// TIA Portal V17 export
// export: Created 2023-03-08T16:44:23.1874801Z, ExportSetting None, DisplayName Totally Integrated Automation Portal, DisplayVersion V17 Update 4, DisplayName TIA Portal Openness, DisplayVersion V17 Update 4, DisplayName TIA Portal Version Control Interface, DisplayVersion V17, DisplayName STEP 7 Professional, DisplayVersion V17 Update 4, DisplayName STEP 7 Safety, DisplayVersion V17, DisplayName WinCC Advanced / Unified PC, DisplayVersion V17 Update 4
DATA_BLOCK "DI"   // DB12
{ S7_Optimized_Access := 'TRUE' }
// stored: AutoNumber false, MemoryReserve 100
   VAR
      LS_045200 : Bool;   // SEPARATOR SUCTION SIDE 1ST. STAGE VERY HIGH LEVEL
      LS_045201 : Bool;   // SEPARATOR SUCTION SIDE 1ST. STAGE VERY LOW LEVEL
      LS_045210 : Bool;   // SEPARATOR DISCHARGE SIDE 1ST. STAGE VERY HIGH
      LS_045211 : Bool;   // SEPARATOR DISCHARGE SIDE 1ST. STAGE VERY LOW
      LS_045220 : Bool;   // SEPARATOR DISCHARGE SIDE 2ND STAGE VERY HIGH
      LS_045221 : Bool;   // SEPARATOR DISCHARGE SIDE 2ND STAGE VERY LOW
      LS_045230 : Bool;   // COALESCER DISCHARGE SIDE 3RD STAGE VERY HIGH
      LS_045232 : Bool;   // COALESCER DISCHARGE SIDE 3RD STAGE VERY LOW
      LS_045240 : Bool;   // OUTLET COALESCER DISCHARGE SIDE 3RD STAGE VERY HIGH
      LS_045242 : Bool;   // OUTLET COALESCER DISCHARGE SIDE 3RD STAGE VERY LOW
      GS_045405 : Bool;   // FLYWHEEL COVER CLOSED
      HS_045009 : Bool;   // EMERGENCY STOP FROM LCP
      HS_045501 : Bool;   // EMERGENCY STOP FROM UCP
      XY_045037 : Bool;   // PROCESS SHUTDOWN FROM DCS
      XY_045035 : Bool;   // EXTERNAL TRIP FROM ESD
      XY_045036 : Bool;   // GAS DETECTION FROM ESD
      LS_045574 : Bool;   // HYDRAULIC OIL VESSEL LOW LEVEL
      LS_045305 : Bool;   // LUBE OIL IN CRANKCASE LOW LEVEL
      LS_045426 : Bool;   // DOWNSTREAM FLOW HEATER LOW LEVEL
      GSH_045206 : Bool;   // BYPASS CONTROL VALVE OVER 1ST-3RD STAGE OPEN
      GSH_045203 : Bool;   // CONDENSATE DRAIN VALVE SEPARATOR SUCTION SIDE 1ST STAGE OPEN
      GSL_045203 : Bool;   // CONDENSATE DRAIN VALVE SEPARATOR SUCTION SIDE 1ST STAGE CLOSED
      GSH_045204 : Bool;   // CONDENSATE DRAIN VALVE SEPARATOR DISCHARGE SIDE 1ST STAGE OPEN
      GSL_045204 : Bool;   // CONDENSATE DRAIN VALVE SEPARATOR DISCHARGE SIDE 1ST STAGE CLOSED
      GSH_045205 : Bool;   // CONDENSATE DRAIN VALVE SEPARATOR DISCHARGE SIDE 2ND STAGE OPEN
      GSL_045205 : Bool;   // CONDENSATE DRAIN VALVE SEPARATOR DISCHARGE SIDE 2ND STAGE CLOSED
      GSH_045207A : Bool;   // CONDENSATE DRAIN VALVE SEPARATOR DISCHARGE SIDE 2ND STAGE OPEN
      GSL_045207A : Bool;   // CONDENSATE DRAIN VALVE SEPARATOR DISCHARGE SIDE 2ND STAGE CLOSED
      GSH_045207B : Bool;   // CONDENSATE DRAIN VALVE SEPARATOR DISCHARGE SIDE 2ND STAGE OPEN
      GSL_045207B : Bool;   // CONDENSATE DRAIN VALVE SEPARATOR DISCHARGE SIDE 2ND STAGE CLOSED
      GSH_045208A : Bool;   // CONDENSATE DRAIN VALVE SEPARATOR DISCHARGE SIDE 3RD STAGE OPEN
      GSL_045208A : Bool;   // CONDENSATE DRAIN VALVE SEPARATOR DISCHARGE SIDE 3RD STAGE CLOSED
      GSH_045208B : Bool;   // CONDENSATE DRAIN VALVE SEPARATOR DISCHARGE SIDE 3RD STAGE OPEN
      GSL_045208B : Bool;   // CONDENSATE DRAIN VALVE SEPARATOR DISCHARGE SIDE 3RD STAGE CLOSED
      TS_045307 : Bool;   // LUBE OIL IN CRANKCASE TEMPERATURE LIMITER
      TC_045306 : Bool;   // LUBE OIL IN CRANKCASE TEMPERATURE CONTROLLER
      TS_045428 : Bool;   // COOLING WATER HEATER TEMPERATURE LIMITER
      TC_045427 : Bool;   // COOLING WATER HEATER TEMPERATURE CONTROLLER
      HS_045001 : Bool;   // COMPRESSOR PREPARE TO START FROM LCP
      HS_045002A : Bool;   // COMPRESSOR PROCESS GAS MODE START FROM LCP
      HS_045002B : Bool;   // COMPRESSOR PROCESS GAS MODE STOP FROM LCP
      HS_045003A : Bool;   // COMPRESSOR NITROGEN MODE START FROM LCP
      HS_045003B : Bool;   // COMPRESSOR NITROGEN MODE STOP FROM LCP
      HS_045004A : Bool;   // CRANKCASE LUBE OIL HEATER START FROM LCP
      HS_045004B : Bool;   // CRANKCASE LUBE OIL HEATER STOP FROM LCP
      HS_045005A : Bool;   // ELECTRICAL OIL PUMP START FROM LCP
      HS_045005B : Bool;   // ELECTRICAL OIL PUMP STOP FROM LCP
      HS_045006A : Bool;   // HYDROCOM HYDRAULIC PUMP START FROM LCP
      HS_045006B : Bool;   // HYDROCOM HYDRAULIC PUMP STOP FROM LCP
      HS_045007A : Bool;   // COMPRESSOR REMOTE FROM LCP
      HS_045007B : Bool;   // COMPRESSOR LOCAL FROM LCP
      HS_045008 : Bool;   // FAULT RESET FROM LCP
      HS_045010 : Bool;   // LAMP TEST FROM LCP
      HS_045011A : Bool;   // COOLANT HEATER START FROM LCP
      HS_045011B : Bool;   // COOLANT HEATER STOP FROM LCP
      HS_045012A : Bool;   // COOLANT PUMP 1 START FROM LCP
      HS_045012B : Bool;   // COOLANT PUMP 1 STOP FROM LCP
      HS_045013A : Bool;   // COOLANT PUMP 2 START FROM LCP
      HS_045013B : Bool;   // COOLANT PUMP 2 STOP FROM LCP
      HS_045014A : Bool;   // FAN 1 START FROM LCP
      HS_045014B : Bool;   // FAN 1 STOP FROM LCP
      HS_045015A : Bool;   // FAN 2 START FROM LCP
      HS_045015B : Bool;   // FAN 2 STOP FROM LCP
      HS_045018A : Bool;   // LOUVER 1 OPEN FROM LCP
      HS_045018B : Bool;   // LOUVER 1 CLOSE FROM LCP
      HS_045019A : Bool;   // LOUVER 2 OPEN FROM LCP
      HS_045019B : Bool;   // LOUVER 2 CLOSE FROM LCP
      HS_045020A : Bool;   // LOUVER 3 OPEN FROM LCP
      HS_045020B : Bool;   // LOUVER 3 CLOSE FROM LCP
      HS_045021A : Bool;   // LOUVER 4 OPEN FROM LCP
      HS_045021B : Bool;   // LOUVER 4 CLOSE FROM LCP
      GSH_045544 : Bool;   // LOUVER 1 OPEN
      GSL_045544 : Bool;   // LOUVER 1 CLOSED
      GSH_045545 : Bool;   // LOUVER 2 OPEN
      GSL_045545 : Bool;   // LOUVER 2 CLOSED
      GSH_045546 : Bool;   // LOUVER 3 OPEN
      GSL_045546 : Bool;   // LOUVER 3 CLOSED
      GSH_045547 : Bool;   // LOUVER 4 OPEN
      GSL_045547 : Bool;   // LOUVER 4 CLOSED
      XY_045001 : Bool;   // OIL HEATER RUNNING FEEDBACK FROM MCC
      XY_045002 : Bool;   // OIL HEATER FAULT FEEDBACK FROM MCC
      XY_045003 : Bool;   // AUXILIARY OIL PUMP RUNNING FEEDBACK FROM MCC
      XY_045004 : Bool;   // AUXILIARY OIL PUMP FAULT FEEDBACK FROM MCC
      XY_045005 : Bool;   // HYDROCOM HYDRAULIC PUMP RUNNING FEEDBACK FROM MCC
      XY_045006 : Bool;   // HYDROCOM HYDRAULIC PUMP FAULT FEEDBACK FROM MCC
      XY_045007 : Bool;   // COOLANT HEATER RUNNING FEEDBACK FROM MCC
      XY_045008 : Bool;   // COOLANT HEATER FAULT FEEDBACK FROM MCC
      XY_045009 : Bool;   // COOLANT PUMP 1 RUNNING FEEDBACK FROM MCC
      XY_045010 : Bool;   // COOLANT PUMP 1 FAULT FEEDBACK FROM MCC
      XY_045011 : Bool;   // COOLANT PUMP 2 RUNNING FEEDBACK FROM MCC
      XY_045012 : Bool;   // COOLANT PUMP 2 FAULT FEEDBACK FROM MCC
      XY_045013 : Bool;   // FAN 1 MOTOR RUNNING FEEDBACK FROM MCC
      XY_045014 : Bool;   // FAN 1 MOTOR FAULT FEEDBACK FROM MCC
      XY_045015 : Bool;   // FAN 2 MOTOR RUNNING FEEDBACK FROM MCC
      XY_045016 : Bool;   // FAN 2 MOTOR FAULT FEEDBACK FROM MCC
      XY_045021 : Bool;   // LOUVER 1 MOTOR RUNNING FEEDBACK FROM MCC
      XY_045022 : Bool;   // LOUVER 1 MOTOR FAULT FEEDBACK FROM MCC
      XY_045023 : Bool;   // LOUVER 2 MOTOR RUNNING FEEDBACK FROM MCC
      XY_045024 : Bool;   // LOUVER 2 MOTOR FAULT FEEDBACK FROM MCC
      XY_045025 : Bool;   // LOUVER 3 MOTOR RUNNING FEEDBACK FROM MCC
      XY_045026 : Bool;   // LOUVER 3 MOTOR FAULT FEEDBACK FROM MCC
      XY_045027 : Bool;   // LOUVER 4 MOTOR RUNNING FEEDBACK FROM MCC
      XY_045028 : Bool;   // LOUVER 4 MOTOR FAULT FEEDBACK FROM MCC
      XY_045029 : Bool;   // COMPRESSOR RUNNING FEEDBACK FROM MV-MCC
      XY_045030 : Bool;   // COMPRESSOR FAULT FEEDBACK FROM MV-MCC
      FS_045540 : Bool;   // AIR OUTLET NOISE ENCLOSURE LOW FLOW
      FS_045541 : Bool;   // AIR OUTLET NOISE ENCLOSURE LOW FLOW
      PDS_045316 : Bool;   // LUBE OIL FILTER POLLUTED
      XY_045033 : Bool;   // CABINET HIGH INTERNAL TEMPERATURE ALARM
      XY_045034 : Bool;   // 24VDC POWER SUPPLY ALARM
      XY_045031 : Bool;   // COMMON ALARM FROM MMS
      XY_045032 : Bool;   // COMMON SHUTDOWN FROM MMS
      UA_045563 : Bool;   // MAINTENANCE FROM CIU
      UA_045562 : Bool;   // ERROR FROM CIU
   END_VAR
BEGIN
END_DATA_BLOCK
